Universal Robots PolyScope program: step5d_strict_rnn_autotune_v3_r022.urp

Program step5d_strict_rnn_autotune_v3_r022 (installation=default directory=/programs/andyl/kunwei/step5 createdIn=5.11.9.1010452 lastSavedIn=5.11.9.1010452 robotSerialNumber=20225200364)
Calibrated DH parameters: a=[0.00002, -0.569483, -0.54992, -0.00001, -0.000036, 0]; d=[0.180894, -146.691669, 192.918669, -46.053088, 0.119778, 0.115602]; alpha=[1.571425, -0.001534, 0.003359, 1.568739, -1.571477, 0]; deltaTheta=[0, 0.376258, -0.101074, -0.275185, -0.000002, 0]
Robot Program (runOnlyOnce=true)
  Script file /programs/andyl/kunwei/step5/step5d_strict_rnn_autotune_v3_r022.script
    | # VERSION: 2026-07-25T163424Z
    | # RELEASE_STAGE_ID: step5d_strict_rnn_autotune_v3_r022
    | # CONTROL_PROFILE_ID: step5d_strict_rnn_autotune_v1
    | # TP_PROGRAM_ID: step5d_strict_rnn_autotune_v3_r022
    | # PHYSICAL_PRIOR_SHA256: c8019aee2c293746e1edb23097aeab1d7dfb1b8dee09df10ce568fb634f47c9f
    | # PARENT_AUTOTUNE_V1_RENDERED_SHA256: eca2c7acaa878b1944c24b46c823ed64ffc0fb9e8658021dfd863a9f624f6676
    | # TP_RUNTIME_IDENTITY_INT: protocol_version=35 digest_hi=36 digest_lo=37
    | global codex_step5d_runtime_protocol_version = 1
    | global codex_step5d_runtime_digest_hi = 1956245643
    | global codex_step5d_runtime_digest_lo = 189200615
    | 
    | def codex_step5d_publish_runtime_identity():
    |   write_output_integer_register(35, codex_step5d_runtime_protocol_version)
    |   write_output_integer_register(36, codex_step5d_runtime_digest_hi)
    |   write_output_integer_register(37, codex_step5d_runtime_digest_lo)
    | end
    | 
    | # Step5d strict RNN ablation v35.
    | # VERSION: 2026-07-15T0204HKT_STEP5D_STRICT_RNN_ABLATION_V35_QUOTA_SAFE_SCHED_OTHER_ACCEL_0P1
    | # GENERATED_AT_LOCAL: 2026-07-15T02:04:25+08:00
    | # ENTRY_XY_M: [0.487795411, 0.129326793]
    | # SAFE_FRAME_SOURCE: config/step5_safe_frame.json from confirmed drag-teach start/mid/end.
    | # NO_SCALE_POLICY: Step5 table frame uses rotation+translation only.
    | # X_GUARD: guard_line=0.488878434 m, path_max_x=0.487795411 m.
    | # TARGET_ROTVEC_RAD: [-3.044172198, -0.130573165, -0.202188631]
    | # PURPOSE: v35 contact search with Stage22/24 gravity-down pre-contact posture, first-contact normal latch, no lift/25.2 attitude cycle and no second contact search, 25.3 bridge deadband acquire into the 5.0-22.0N filtered preload window with 3.0-25.0N raw sanity and bridge-time preload parameter channel, 25.95 register clear barrier, then v35 Step5d ablation Stage25.0 layout-524-only speedj strict RNN live candidate for 60 s.
    | # FLOW_TABLE: STEP5_FLOW.md
    | # STEP5_STAGE_ID: step5d_strict_rnn_autotune_v3
    | # PARENT_V35_SHA256: 50894de5cdf74dd17309c829b904251a3da26613a4d73e93653f7c165f5fbbd0
    | # STEP5_TABLE_SOURCE: config/step5_stage_table.json
    | # TP_ROLE: layout524_speedj_executor_and_structural_guard_only; Step5d v35 accepts only bridge-computed strict RNN qdot; marker 524 is internal to the Stage25 joint packet.
    | # REGISTER_CONTRACT: Stage 25.3 is a no-motion structural handoff. Stage 25.95 requires bridge-cleared registers 37..47 before Stage 25.0. Stage 25.0 accepts only register 47=524.0; registers 37..42 are strict RNN qd0..qd5, 43 cmd_valid, 44 path_time_s. Layout 523.0 and Cartesian/DLS runtime commands are forbidden.
    | # PRECONTACT_POSE_CONTRACT: config/step_pose_contract_table.json pre_contact_search_gravity_down_v1; Stage22/24 TCP +Z targets base -Z using [pi,0,0].
    | # STAGE25_CONTACT_SAFETY: v35 bridge keeps 60N normal/100N force guards and 3.0Nm torque guard; speedj_rnn_live is the only future live command source; speedl_cartesian_oracle and speedj_dls_oracle are offline shadow/diagnostic only and must never be sent as runtime fallback.
    | # FORCE_FRAME_CONTRACT: UR_FORCE_FRAME_CONTRACT.md; reaction normal for load, approach normal for posture.
    | # STAGE25_V35_SCAFFOLD: v31_permissive_contact_frame_contract_layout524_60s
    | # STEP5_PATH_FORMULA: Step5 table stage step5_contact_cycloid_baseline_v1: local-basis x=0.015 * (0.1t - sin(0.1t)), y=0.015 * (1 - cos(0.1t)), duration=60s
    | # FIRST_CONTACT_Z_EVIDENCE: bridge_step4e_line_outerloop_v13_autowatch_20260609_141027 force jump at z=0.008044839 m; v16 cross-check z=0.007996174 m.
    | # AUTOTUNE_CONTROL: fixed tau=.35s, fixed dt=.002s, profile rate .010/.015/.020; normal_filter_alpha is not an active candidate dimension.
    | # SAFETY: raw normal guard 60 N, force norm guard 100 N, torque guard 3.0 Nm.
    | 
    | def codex_abs(x):
    |   if x < 0.0:
    |     return -x
    |   end
    |   return x
    | end
    | 
    | def codex_clamp(x, lo, hi):
    |   if x < lo:
    |     return lo
    |   elif x > hi:
    |     return hi
    |   end
    |   return x
    | end
    | 
    | def codex_wait_for_fresh_heartbeat(timeout_s):
    |   local t = 0.0
    |   local initial_heartbeat = read_input_float_register(26)
    |   local current_heartbeat = initial_heartbeat
    |   while t < timeout_s:
    |     current_heartbeat = read_input_float_register(26)
    |     write_output_float_register(26, current_heartbeat)
    |     if read_input_float_register(27) > 0.5 and current_heartbeat != initial_heartbeat:
    |       return True
    |     end
    |     sync()
    |     t = t + get_steptime()
    |   end
    |   return False
    | end
    | 
    | def codex_wait_for_rezero_complete(timeout_s):
    |   local t = 0.0
    |   local initial_heartbeat = read_input_float_register(26)
    |   local current_heartbeat = initial_heartbeat
    |   local saw_sensor_not_ready = False
    |   while t < timeout_s:
    |     current_heartbeat = read_input_float_register(26)
    |     write_output_float_register(26, current_heartbeat)
    |     if read_input_float_register(27) < 0.5:
    |       saw_sensor_not_ready = True
    |     elif saw_sensor_not_ready and read_input_float_register(27) > 0.5 and current_heartbeat != initial_heartbeat:
    |       return True
    |     end
    |     sync()
    |     t = t + get_steptime()
    |   end
    |   return False
    | end
    | 
    | def codex_step4e_guard_stop_reason():
    |   local normal_force = read_input_float_register(24)
    |   local force_norm = read_input_float_register(25)
    |   local sensor_ok = read_input_float_register(27)
    |   local stop_request = read_input_float_register(28)
    |   local torque_norm = read_input_float_register(30)
    |   if sensor_ok < 0.5:
    |     return 3.0
    |   elif stop_request > 0.5:
    |     return 4.0
    |   elif codex_abs(normal_force) > 60.0:
    |     return 5.0
    |   elif force_norm > 100.0:
    |     return 6.0
    |   elif torque_norm > 3.0:
    |     return 7.0
    |   end
    |   return 0.0
    | end
    | 
    | def codex_should_auto_home(stop_reason):
    |   if stop_reason == 1.0:
    |     return True
    |   elif stop_reason == 2.0:
    |     # Transport/heartbeat loss may follow a protective stop; never auto-home.
    |     return False
    |   elif stop_reason == 4.0:
    |     return True
    |   elif stop_reason == 5.0:
    |     return True
    |   elif stop_reason == 6.0:
    |     return True
    |   elif stop_reason == 7.0:
    |     return True
    |   elif stop_reason == 8.0:
    |     return True
    |   elif stop_reason == 9.0:
    |     return True
    |   elif stop_reason == 10.0:
    |     return True
    |   elif stop_reason == 12.0:
    |     return True
    |   elif stop_reason == 13.0:
    |     return True
    |   elif stop_reason == 14.0:
    |     return True
    |   elif stop_reason == 17.0:
    |     # Reserved unsafe-entry/safety interruption reason; never auto-home.
    |     return False
    |   end
    |   return False
    | end
    | 
    | def codex_echo_basic(stop_reason):
    |   write_output_float_register(24, read_input_float_register(24))
    |   write_output_float_register(25, read_input_float_register(25))
    |   write_output_float_register(26, read_input_float_register(26))
    |   write_output_float_register(27, read_input_float_register(27))
    |   write_output_float_register(28, read_input_float_register(28))
    |   write_output_float_register(29, read_input_float_register(29))
    |   write_output_float_register(30, stop_reason)
    | end
    | 
    | def codex_echo_step4e(stop_reason):
    |   codex_echo_basic(stop_reason)
    |   write_output_float_register(31, read_input_float_register(44))
    |   write_output_float_register(32, read_input_float_register(45))
    |   write_output_float_register(33, read_input_float_register(39))
    |   write_output_float_register(36, read_input_float_register(37))
    |   write_output_float_register(37, read_input_float_register(38))
    |   write_output_float_register(38, read_input_float_register(39))
    |   write_output_float_register(39, read_input_float_register(40))
    |   write_output_float_register(40, read_input_float_register(41))
    |   write_output_float_register(41, read_input_float_register(42))
    |   write_output_float_register(42, read_input_float_register(43))
    |   write_output_float_register(43, read_input_float_register(44))
    |   write_output_float_register(44, read_input_float_register(45))
    |   write_output_float_register(45, read_input_float_register(46))
    |   write_output_float_register(46, read_input_float_register(47))
    | end
    | 
    | 
    | def codex_wait_for_cmd_valid(stage_code, timeout_s):
    |   local t = 0.0
    |   local last_heartbeat = read_input_float_register(26)
    |   local stale_s = 0.0
    |   while t < timeout_s:
    |     write_output_float_register(35, stage_code)
    |     local heartbeat = read_input_float_register(26)
    |     if heartbeat == last_heartbeat:
    |       stale_s = stale_s + get_steptime()
    |     else:
    |       stale_s = 0.0
    |       last_heartbeat = heartbeat
    |     end
    |     codex_echo_step4e(0.0)
    |     if stale_s > 0.100:
    |       return 2.0
    |     end
    |     local guard_reason = codex_step4e_guard_stop_reason()
    |     if guard_reason != 0.0:
    |       return guard_reason
    |     end
    |     if read_input_float_register(43) >= 0.5:
    |       return 0.0
    |     end
    |     sync()
    |     t = t + get_steptime()
    |   end
    |   return 12.0
    | end
    | 
    | 
    | def codex_wait_for_stage_linear_zero(stage_code, timeout_s):
    |   local t = 0.0
    |   local last_heartbeat = read_input_float_register(26)
    |   local stale_s = 0.0
    |   while t < timeout_s:
    |     write_output_float_register(35, stage_code)
    |     local heartbeat = read_input_float_register(26)
    |     if heartbeat == last_heartbeat:
    |       stale_s = stale_s + get_steptime()
    |     else:
    |       stale_s = 0.0
    |       last_heartbeat = heartbeat
    |     end
    |     codex_echo_step4e(0.0)
    |     if stale_s > 0.100:
    |       return 2.0
    |     end
    |     local guard_reason = codex_step4e_guard_stop_reason()
    |     if guard_reason != 0.0:
    |       return guard_reason
    |     end
    |     if read_input_float_register(43) >= 0.5 and codex_abs(read_input_float_register(37)) <= 0.000001 and codex_abs(read_input_float_register(38)) <= 0.000001 and codex_abs(read_input_float_register(39)) <= 0.000001:
    |       return 0.0
    |     end
    |     sync()
    |     t = t + get_steptime()
    |   end
    |   return 12.0
    | end
    | 
    | def codex_step5d_down_search(search_stage, near_stage, max_search_down_m, search_near_start_depth_m, search_runtime_limit_s, search_far_speed_m_s, search_near_speed_m_s):
    |   local stop_reason = 0.0
    |   local search_accel_m_s2 = 0.300
    |   local search_hold_s = 0.002
    |   local stale_limit_s = 0.100
    |   local search_start = get_actual_tcp_pose()
    |   local last_heartbeat = read_input_float_register(26)
    |   local stale_s = 0.0
    |   local t = 0.0
    |   while stop_reason == 0.0:
    |     local heartbeat = read_input_float_register(26)
    |     local normal_force = read_input_float_register(24)
    |     local force_norm = read_input_float_register(25)
    |     local pose_now = get_actual_tcp_pose()
    |     local search_depth_m = search_start[2] - pose_now[2]
    |     if heartbeat == last_heartbeat:
    |       stale_s = stale_s + get_steptime()
    |     else:
    |       stale_s = 0.0
    |       last_heartbeat = heartbeat
    |     end
    |     if normal_force <= -1.0 or force_norm > 1.5:
    |       stop_reason = 11.0
    |       if search_depth_m < search_near_start_depth_m:
    |         write_output_float_register(35, search_stage)
    |       else:
    |         write_output_float_register(35, near_stage)
    |       end
    |       codex_echo_step4e(stop_reason)
    |     elif stale_s > stale_limit_s:
    |       stop_reason = 2.0
    |     else:
    |       stop_reason = codex_step4e_guard_stop_reason()
    |     end
    |     if stop_reason == 0.0:
    |       if search_depth_m >= max_search_down_m:
    |         stop_reason = 8.0
    |       elif t >= search_runtime_limit_s:
    |         stop_reason = 10.0
    |       else:
    |         if search_depth_m < search_near_start_depth_m:
    |           write_output_float_register(35, search_stage)
    |           codex_echo_step4e(stop_reason)
    |           speedl([0.0, 0.0, search_far_speed_m_s, 0.0, 0.0, 0.0], search_accel_m_s2, search_hold_s)
    |         else:
    |           write_output_float_register(35, near_stage)
    |           codex_echo_step4e(stop_reason)
    |           speedl([0.0, 0.0, search_near_speed_m_s, 0.0, 0.0, 0.0], search_accel_m_s2, search_hold_s)
    |         end
    |         t = t + get_steptime()
    |       end
    |     end
    |   end
    |   stopl(0.1)
    |   return stop_reason
    | end
    | 
    | def codex_step5d_autotune_trial_v1(campaign_home_pose, tp_speedj_accel_rad_s2, batch_row_index):
    |   local stop_reason = 0.0
    |   local home_pose = campaign_home_pose
    |   local entry_x = 0.487834547
    |   local entry_y = 0.129337053
    |   local precontact_z = 0.022863519
    |   local minimum_start_above_entry_m = 0.010000000
    |   # PRECONTACT_POSE_PRIOR_ID: step5d_v3_physical_prior_contact_0p1_20260719; completed contact-plus-0.1s robust pose plus clearance before guarded search.
    |   local target_rx = 3.120752062
    |   local target_ry = 0.000000000
    |   local target_rz = 0.068626833
    |   local line_accel_m_s2 = 0.300
    |   local line_hold_s = 0.002
    |   local line_runtime_limit_s = 75.000
    |   local line_success_progress_m = 60.000000000
    |   local end_hold_required_s = 0.100
    |   local end_hold_s = 0.0
    |   local max_cmd_angular_xy_rad_s = 0.120
    |   local cmd_valid_grace_s = 0.250
    |   local cmd_valid_loss_limit_s = 0.100
    |   local cmd_invalid_s = 0.0
    |   local saw_cmd_valid = 0
    |   local short_retract_z_m = 0.010
    |   local short_retract_speed_m_s = 0.040
    |   local home_return_speed_m_s = 0.050
    |   local final_progress_m = 0.0
    | 
    |   textmsg("codex step4e version 2026-07-15T0204HKT_STEP5D_STRICT_RNN_ABLATION_V35_QUOTA_SAFE_SCHED_OTHER_ACCEL_0P1 start step5d_strict_rnn_ablation_v35")
    |   write_output_float_register(34, 0.0)
    |   write_output_float_register(35, 20.0)
    |   codex_echo_step4e(0.0)
    |   if not codex_wait_for_fresh_heartbeat(60.0):
    |     stop_reason = 3.0
    |   end
    | 
    |   if stop_reason == 0.0:
    |     local p_current = get_actual_tcp_pose()
    |     local expected_home_orientation = p[p_current[0], p_current[1], p_current[2], target_rx, target_ry, target_rz]
    |     local home_orientation_delta = pose_trans(pose_inv(expected_home_orientation), p_current)
    |     local home_orientation_error_rad = sqrt(home_orientation_delta[3] * home_orientation_delta[3] + home_orientation_delta[4] * home_orientation_delta[4] + home_orientation_delta[5] * home_orientation_delta[5])
    |     if p_current[2] < precontact_z + minimum_start_above_entry_m or home_orientation_error_rad > 0.035:
    |       return 17.0
    |     else:
    |       write_output_float_register(35, 22.0)
    |       local entry_xy_pose = p[entry_x, entry_y, p_current[2], target_rx, target_ry, target_rz]
    |       local entry_precontact_pose = p[entry_x, entry_y, precontact_z, target_rx, target_ry, target_rz]
    |       codex_echo_step4e(stop_reason)
    |       movel(entry_xy_pose, a=0.135, v=0.090, r=0.0)
    |       stopl(0.1)
    |       movel(entry_precontact_pose, a=0.060, v=0.040, r=0.0)
    |       stopl(0.1)
    |       sleep(0.20)
    |     end
    |     write_output_float_register(35, 23.0)
    |     codex_echo_step4e(stop_reason)
    |     write_output_float_register(34, 1.0)
    |     if not codex_wait_for_rezero_complete(5.0):
    |       stop_reason = 14.0
    |     end
    |     if stop_reason == 0.0:
    |       sleep(0.20)
    |       stop_reason = codex_step4e_guard_stop_reason()
    |     end
    |   end
    | 
    |   if stop_reason == 0.0:
    |     local first_contact_z_m = 0.008044839
    |     local first_near_start_z_m = first_contact_z_m + 0.020
    |     local first_max_end_z_m = first_contact_z_m - 0.004
    |     local first_search_start_pose = get_actual_tcp_pose()
    |     local first_search_near_start_depth_m = first_search_start_pose[2] - first_near_start_z_m
    |     local first_search_max_down_m = first_search_start_pose[2] - first_max_end_z_m
    |     if first_search_near_start_depth_m < 0.0:
    |       first_search_near_start_depth_m = 0.0
    |     end
    |     if first_search_max_down_m < 0.020:
    |       first_search_max_down_m = 0.020
    |     end
    |     if first_search_max_down_m < first_search_near_start_depth_m + 0.010:
    |       first_search_max_down_m = first_search_near_start_depth_m + 0.010
    |     end
    |     stop_reason = codex_step5d_down_search(24.0, 24.2, first_search_max_down_m, first_search_near_start_depth_m, 40.000, -0.03375, -0.0025)
    |     if stop_reason == 11.0:
    |       stop_reason = 0.0
    |     end
    |   end
    | 
    |   if stop_reason == 0.0:
    |     write_output_float_register(35, 25.05)
    |     stop_reason = codex_wait_for_cmd_valid(25.05, 1.000)
    |   end
    | 
    |   if stop_reason == 0.0:
    |     write_output_float_register(35, 25.15)
    |     codex_echo_step4e(stop_reason)
    |     sync()
    |   end
    | 
    |   if stop_reason == 0.0:
    |     write_output_float_register(35, 25.3)
    |     local last_heartbeat_entry = read_input_float_register(26)
    |     local stale_s_entry = 0.0
    |     local t_entry = 0.0
    |     local line_entry_s = 0.0
    |     local line_entry_default_required_s = 0.000
    |     local line_entry_default_timeout_s = 60.000
    |     local line_entry_default_normal_load_min_n = 5.000
    |     local line_entry_default_normal_load_max_n = 22.000
    |     local line_entry_default_force_norm_max_n = 100.000
    |     local line_entry_recovery_normal_load_min_n = 0.000
    |     local line_entry_recovery_normal_load_max_n = 100.000
    |     local line_entry_force_norm_stop_n = 100.000
    |     local line_entry_cmd_limit_m_s = 0.003
    |     local line_entry_param_valid_code = 521.000
    |     saw_cmd_valid = 0
    |     cmd_invalid_s = 0.0
    |     while stop_reason == 0.0:
    |       local heartbeat_entry = read_input_float_register(26)
    |       local cmd_valid = read_input_float_register(43)
    |       local cmd_vx = read_input_float_register(37)
    |       local cmd_vy = read_input_float_register(38)
    |       local cmd_vz = read_input_float_register(39)
    |       local target_force = read_input_float_register(29)
    |       local force_error = read_input_float_register(45)
    |       local normal_load = target_force - force_error
    |       local force_norm = read_input_float_register(25)
    |       local loop_dt = get_steptime()
    |       local line_entry_required_s = line_entry_default_required_s
    |       local line_entry_timeout_s = line_entry_default_timeout_s
    |       local line_entry_normal_load_min_n = line_entry_default_normal_load_min_n
    |       local line_entry_normal_load_max_n = line_entry_default_normal_load_max_n
    |       local line_entry_force_norm_max_n = line_entry_default_force_norm_max_n
    |       local line_entry_param_valid = read_input_float_register(47)
    |       if codex_abs(line_entry_param_valid - line_entry_param_valid_code) < 0.001:
    |         local candidate_min_n = read_input_float_register(40)
    |         local candidate_max_n = read_input_float_register(41)
    |         local candidate_force_norm_max_n = read_input_float_register(42)
    |         local candidate_required_s = read_input_float_register(44)
    |         local candidate_timeout_s = read_input_float_register(46)
    |         if candidate_min_n >= 0.0 and candidate_max_n >= candidate_min_n and candidate_force_norm_max_n > 0.0 and candidate_force_norm_max_n <= line_entry_force_norm_stop_n and candidate_required_s >= 0.0 and candidate_timeout_s > candidate_required_s:
    |           line_entry_normal_load_min_n = candidate_min_n
    |           line_entry_normal_load_max_n = candidate_max_n
    |           line_entry_force_norm_max_n = candidate_force_norm_max_n
    |           line_entry_required_s = candidate_required_s
    |           line_entry_timeout_s = candidate_timeout_s
    |         end
    |       end
    |       if cmd_valid >= 0.5:
    |         saw_cmd_valid = 1
    |         cmd_invalid_s = 0.0
    |       else:
    |         cmd_invalid_s = cmd_invalid_s + loop_dt
    |       end
    |       if heartbeat_entry == last_heartbeat_entry:
    |         stale_s_entry = stale_s_entry + loop_dt
    |       else:
    |         stale_s_entry = 0.0
    |         last_heartbeat_entry = heartbeat_entry
    |       end
    |       t_entry = t_entry + loop_dt
    |       if cmd_valid >= 0.5:
    |         line_entry_s = line_entry_s + loop_dt
    |       else:
    |         line_entry_s = 0.0
    |       end
    |       codex_echo_step4e(stop_reason)
    |       if stale_s_entry > 1.000:
    |         stop_reason = 2.0
    |       else:
    |         stop_reason = codex_step4e_guard_stop_reason()
    |       end
    |       if stop_reason == 0.0:
    |         if line_entry_s >= line_entry_required_s:
    |           stop_reason = 16.0
    |         elif cmd_valid < 0.5:
    |           if saw_cmd_valid == 0 and t_entry < cmd_valid_grace_s:
    |             sync()
    |           elif saw_cmd_valid == 1 and cmd_invalid_s <= cmd_valid_loss_limit_s:
    |             sync()
    |           else:
    |             stop_reason = 12.0
    |           end
    |         elif t_entry >= line_entry_timeout_s:
    |           stop_reason = 12.0
    |         else:
    |           sync()
    |         end
    |       end
    |     end
    |     stopl(0.1)
    |     if stop_reason == 16.0:
    |       stop_reason = 0.0
    |       saw_cmd_valid = 0
    |       cmd_invalid_s = 0.0
    |       end_hold_s = 0.0
    |       write_output_float_register(35, 25.95)
    |       local register_clear_required_s = 0.006
    |       local register_clear_timeout_s = 1.000
    |       local register_clear_s = 0.0
    |       local register_clear_t = 0.0
    |       local register_clear_zero_tol = 0.000500
    |       local last_heartbeat_clear = read_input_float_register(26)
    |       local stale_s_clear = 0.0
    |       while stop_reason == 0.0 and register_clear_s < register_clear_required_s and register_clear_t < register_clear_timeout_s:
    |         local heartbeat_clear = read_input_float_register(26)
    |         local clear_cmd_valid = read_input_float_register(43)
    |         local clear_reg0 = read_input_float_register(37)
    |         local clear_reg1 = read_input_float_register(38)
    |         local clear_reg2 = read_input_float_register(39)
    |         local clear_reg3 = read_input_float_register(40)
    |         local clear_reg4 = read_input_float_register(41)
    |         local clear_reg5 = read_input_float_register(42)
    |         local clear_layout_tag = read_input_float_register(47)
    |         local loop_dt = get_steptime()
    |         if heartbeat_clear == last_heartbeat_clear:
    |           stale_s_clear = stale_s_clear + loop_dt
    |         else:
    |           stale_s_clear = 0.0
    |           last_heartbeat_clear = heartbeat_clear
    |         end
    |         register_clear_t = register_clear_t + loop_dt
    |         codex_echo_step4e(stop_reason)
    |         if stale_s_clear > 1.000:
    |           stop_reason = 2.0
    |         else:
    |           stop_reason = codex_step4e_guard_stop_reason()
    |         end
    |         if stop_reason == 0.0:
    |           if clear_cmd_valid < 0.5 and codex_abs(clear_layout_tag - line_entry_param_valid_code) >= 0.001 and codex_abs(clear_layout_tag - 523.000) >= 0.001 and codex_abs(clear_layout_tag - 524.000) >= 0.001 and codex_abs(clear_reg0) <= register_clear_zero_tol and codex_abs(clear_reg1) <= register_clear_zero_tol and codex_abs(clear_reg2) <= register_clear_zero_tol and codex_abs(clear_reg3) <= register_clear_zero_tol and codex_abs(clear_reg4) <= register_clear_zero_tol and codex_abs(clear_reg5) <= register_clear_zero_tol:
    |             register_clear_s = register_clear_s + loop_dt
    |           else:
    |             register_clear_s = 0.0
    |           end
    |           sync()
    |         end
    |       end
    |       if stop_reason == 0.0 and register_clear_s < register_clear_required_s:
    |         stop_reason = 12.0
    |       end
    |     end
    |   end
    | 
    |   if stop_reason == 0.0:
    |     write_output_float_register(35, 25.0)
    |     local last_heartbeat2 = read_input_float_register(26)
    |     local stale_s2 = 0.0
    |     local t2 = 0.0
    |     local qdot_cap_rad_s = 0.500
    |     local cartesian_linear_cap_m_s = 1.000
    |     local cartesian_angular_cap_rad_s = 1.000
    |     local cartesian_accel_m_s2 = 0.050
    |     local joint_accel_rad_s2 = tp_speedj_accel_rad_s2
    |     local cartesian_layout_code = 523.000
    |     local joint_layout_code = 524.000
    |     local stage25_have_accepted_command = False
    |     # STAGE25_CADENCE_CONSUMPTION: output register 47 is 1 only when this
    |     # TP loop accepts a current Stage25 command packet and reaches speedl/speedj.
    |     while stop_reason == 0.0:
    |       local heartbeat2 = read_input_float_register(26)
    |       local cmd_valid = read_input_float_register(43)
    |       local progress_s = read_input_float_register(44)
    |       local stage25_layout_tag = read_input_float_register(47)
    |       local stage25_command_consumed = 0
    |       local cartesian_layout_ok = codex_abs(stage25_layout_tag - cartesian_layout_code) < 0.001
    |       local joint_layout_ok = codex_abs(stage25_layout_tag - joint_layout_code) < 0.001
    |       local cmd_qd0 = read_input_float_register(37)
    |       local cmd_qd1 = read_input_float_register(38)
    |       local cmd_qd2 = read_input_float_register(39)
    |       local cmd_qd3 = read_input_float_register(40)
    |       local cmd_qd4 = read_input_float_register(41)
    |       local cmd_qd5 = read_input_float_register(42)
    |       local cmd_vx = cmd_qd0
    |       local cmd_vy = cmd_qd1
    |       local cmd_vz = cmd_qd2
    |       local cmd_wx = cmd_qd3
    |       local cmd_wy = cmd_qd4
    |       local cmd_wz = cmd_qd5
    |       local loop_dt = get_steptime()
    |       local heartbeat_fresh = False
    |       final_progress_m = progress_s
    |       if cmd_valid >= 0.5 and joint_layout_ok:
    |         saw_cmd_valid = 1
    |         cmd_invalid_s = 0.0
    |       else:
    |         cmd_invalid_s = cmd_invalid_s + loop_dt
    |       end
    |       if heartbeat2 == last_heartbeat2:
    |         stale_s2 = stale_s2 + loop_dt
    |       else:
    |         stale_s2 = 0.0
    |         last_heartbeat2 = heartbeat2
    |         heartbeat_fresh = True
    |       end
    |       t2 = t2 + loop_dt
    |       if progress_s >= line_success_progress_m:
    |         end_hold_s = end_hold_s + loop_dt
    |       else:
    |         end_hold_s = 0.0
    |       end
    |       codex_echo_step4e(stop_reason)
    |       if stale_s2 > 1.000:
    |         stop_reason = 2.0
    |       else:
    |         stop_reason = codex_step4e_guard_stop_reason()
    |       end
    |       if stop_reason == 0.0:
    |         # DEADLINE_OVERRUN_LAST_COMMAND_HOLD: bounded zero-order hold.
    |         if not heartbeat_fresh:
    |           if stage25_have_accepted_command and cmd_valid >= 0.5 and joint_layout_ok and codex_abs(cmd_qd0) <= qdot_cap_rad_s and codex_abs(cmd_qd1) <= qdot_cap_rad_s and codex_abs(cmd_qd2) <= qdot_cap_rad_s and codex_abs(cmd_qd3) <= qdot_cap_rad_s and codex_abs(cmd_qd4) <= qdot_cap_rad_s and codex_abs(cmd_qd5) <= qdot_cap_rad_s:
    |             stage25_command_consumed = 1
    |             write_output_float_register(47, stage25_command_consumed)
    |             speedj([cmd_qd0, cmd_qd1, cmd_qd2, cmd_qd3, cmd_qd4, cmd_qd5], joint_accel_rad_s2, line_hold_s)
    |           else:
    |             write_output_float_register(47, stage25_command_consumed)
    |             sync()
    |           end
    |         elif cmd_valid < 0.5 or not joint_layout_ok:
    |           write_output_float_register(47, stage25_command_consumed)
    |           if saw_cmd_valid == 0 and t2 < cmd_valid_grace_s:
    |             sync()
    |           elif saw_cmd_valid == 1 and cmd_invalid_s <= cmd_valid_loss_limit_s:
    |             sync()
    |           else:
    |             stop_reason = 12.0
    |           end
    |         elif joint_layout_ok and (codex_abs(cmd_qd0) > qdot_cap_rad_s or codex_abs(cmd_qd1) > qdot_cap_rad_s or codex_abs(cmd_qd2) > qdot_cap_rad_s or codex_abs(cmd_qd3) > qdot_cap_rad_s or codex_abs(cmd_qd4) > qdot_cap_rad_s or codex_abs(cmd_qd5) > qdot_cap_rad_s):
    |           write_output_float_register(47, stage25_command_consumed)
    |           stop_reason = 13.0
    |         elif end_hold_s >= end_hold_required_s:
    |           write_output_float_register(47, stage25_command_consumed)
    |           stop_reason = 1.0
    |         elif t2 >= line_runtime_limit_s:
    |           write_output_float_register(47, stage25_command_consumed)
    |           stop_reason = 10.0
    |         else:
    |           stage25_have_accepted_command = True
    |           stage25_command_consumed = 1
    |           write_output_float_register(47, stage25_command_consumed)
    |           speedj([cmd_qd0, cmd_qd1, cmd_qd2, cmd_qd3, cmd_qd4, cmd_qd5], joint_accel_rad_s2, line_hold_s)
    |         end
    |       end
    |     end
    |     stopj(0.3)
    |     stopl(0.1)
    |   end
    | 
    |   write_output_float_register(30, stop_reason)
    |   write_output_float_register(31, final_progress_m)
    |   write_output_float_register(35, 29.0)
    |   textmsg("codex step4e version 2026-07-15T0204HKT_STEP5D_STRICT_RNN_ABLATION_V35_QUOTA_SAFE_SCHED_OTHER_ACCEL_0P1 stop reason:", stop_reason)
    |   return stop_reason
    | end
    | 
    | # STEP5D_AUTOTUNE_CONTINUOUS_TP: every trial returns to the captured campaign home.
    | # Immutable bundle cold-read precedes each rolling next ARM; no ACK command is active.
    | # HOST_TO_TP_INT: epoch=24 trial=25 command=26 token=27 profile=28 sequence=29 batch_row=30 logical_batch=31
    | # TP_TO_HOST_INT: epoch=24 trial=25 state=26 token=27 reason=28 profile=29 consumed_sequence=30 batch_row=31 return_kind=32 guard_mask=33 logical_batch=34
    | # PROFILE_ID: hundreds=normal-rate level; tens=host-slew level; ones=TP accel level
    | # NETWORK_PROFILE_LEVELS: normal=1..3 (.010/.015/.020); host/TP=1..3 (.1/.2/.5)
    | # PROFILE_NORMAL_LEVELS: 1=.010, 2=.015, 3=.020, 5=.050, 6=.100 rad/s;
    | # level 4 (.030 rad/s) is offline_only and must never reach this TP
    | # TP_ACCEL_LEVEL: 1=.1 rad/s^2, 2=.2 rad/s^2, 3=.5 rad/s^2
    | # STOP_CONTRACT: integer STOP is polled only in stationary ready states; during RUN
    | # the frozen trial consumes the legacy float stop_request safety carrier.
    | 
    | global codex_autotune_batch_row_echo = 0
    | global codex_autotune_return_kind_echo = 0
    | global codex_autotune_return_guard_mask = 0
    | global codex_autotune_return_observer_active = False
    | global codex_autotune_return_segment_id = 0
    | global codex_autotune_return_current_angular_speed_rad_s = 0.0
    | global codex_autotune_return_current_angular_accel_rad_s2 = 0.0
    | global codex_autotune_return_max_angular_speed_rad_s = 0.0
    | global codex_autotune_return_max_angular_accel_rad_s2 = 0.0
    | global codex_autotune_return_max_sample_gap_s = 0.0
    | global codex_autotune_logical_batch_sequence_echo = 0
    | 
    | def codex_autotune_norm3(x, y, z):
    |   return sqrt(x * x + y * y + z * z)
    | end
    | 
    | thread codex_autotune_return_telemetry_observer():
    |   local have_controller_time_sample = False
    |   local have_angular_sample = False
    |   local last_wx = 0.0
    |   local last_wy = 0.0
    |   local last_wz = 0.0
    |   local controller_clock = time()
    |   local last_controller_time_s = controller_clock.sec + controller_clock.nanosec / 1000000000.0
    |   while codex_autotune_return_observer_active:
    |     controller_clock = time()
    |     local controller_time_s = controller_clock.sec + controller_clock.nanosec / 1000000000.0
    |     local loop_dt = controller_time_s - last_controller_time_s
    |     last_controller_time_s = controller_time_s
    |     local tcp_speed = get_actual_tcp_speed()
    |     local angular_speed_rad_s = codex_autotune_norm3(tcp_speed[3], tcp_speed[4], tcp_speed[5])
    |     local angular_accel_rad_s2 = 0.0
    |     if have_controller_time_sample and have_angular_sample and loop_dt > 0.0:
    |       local angular_filter_alpha = loop_dt / (0.020 + loop_dt)
    |       local filtered_wx = last_wx + angular_filter_alpha * (tcp_speed[3] - last_wx)
    |       local filtered_wy = last_wy + angular_filter_alpha * (tcp_speed[4] - last_wy)
    |       local filtered_wz = last_wz + angular_filter_alpha * (tcp_speed[5] - last_wz)
    |       angular_accel_rad_s2 = codex_autotune_norm3(filtered_wx - last_wx, filtered_wy - last_wy, filtered_wz - last_wz) / loop_dt
    |       last_wx = filtered_wx
    |       last_wy = filtered_wy
    |       last_wz = filtered_wz
    |     else:
    |       last_wx = tcp_speed[3]
    |       last_wy = tcp_speed[4]
    |       last_wz = tcp_speed[5]
    |     end
    |     have_angular_sample = True
    |     codex_autotune_return_current_angular_speed_rad_s = angular_speed_rad_s
    |     codex_autotune_return_current_angular_accel_rad_s2 = angular_accel_rad_s2
    |     if angular_speed_rad_s > codex_autotune_return_max_angular_speed_rad_s:
    |       codex_autotune_return_max_angular_speed_rad_s = angular_speed_rad_s
    |     end
    |     if angular_accel_rad_s2 > codex_autotune_return_max_angular_accel_rad_s2:
    |       codex_autotune_return_max_angular_accel_rad_s2 = angular_accel_rad_s2
    |     end
    |     if have_controller_time_sample and loop_dt > codex_autotune_return_max_sample_gap_s:
    |       codex_autotune_return_max_sample_gap_s = loop_dt
    |     end
    |     have_controller_time_sample = True
    |     sync()
    |   end
    | end
    | 
    | def codex_autotune_latch_return_telemetry():
    |   write_output_float_register(35, 40.3)
    |   write_output_float_register(39, 3.0)
    |   write_output_float_register(40, codex_autotune_return_current_angular_speed_rad_s)
    |   write_output_float_register(41, codex_autotune_return_current_angular_accel_rad_s2)
    |   write_output_float_register(42, codex_autotune_return_max_angular_speed_rad_s)
    |   write_output_float_register(43, codex_autotune_return_max_angular_accel_rad_s2)
    |   write_output_float_register(44, codex_autotune_return_max_sample_gap_s)
    | end
    | 
    | def codex_autotune_typed_target_verified(target_pose, campaign_home_q, require_home_q):
    |   local actual_pose = get_actual_tcp_pose()
    |   local delta_pose = pose_trans(pose_inv(target_pose), actual_pose)
    |   local position_error_m = sqrt(delta_pose[0] * delta_pose[0] + delta_pose[1] * delta_pose[1] + delta_pose[2] * delta_pose[2])
    |   local orientation_error_rad = sqrt(delta_pose[3] * delta_pose[3] + delta_pose[4] * delta_pose[4] + delta_pose[5] * delta_pose[5])
    |   local tcp_speed = get_actual_tcp_speed()
    |   local linear_speed_m_s = sqrt(tcp_speed[0] * tcp_speed[0] + tcp_speed[1] * tcp_speed[1] + tcp_speed[2] * tcp_speed[2])
    |   local angular_speed_rad_s = sqrt(tcp_speed[3] * tcp_speed[3] + tcp_speed[4] * tcp_speed[4] + tcp_speed[5] * tcp_speed[5])
    |   local actual_qd = get_actual_joint_speeds()
    |   local qd_max_rad_s = 0.0
    |   local qd_index = 0
    |   while qd_index < 6:
    |     if codex_abs(actual_qd[qd_index]) > qd_max_rad_s:
    |       qd_max_rad_s = codex_abs(actual_qd[qd_index])
    |     end
    |     qd_index = qd_index + 1
    |   end
    |   local home_q_ok = True
    |   if require_home_q:
    |     home_q_ok = codex_autotune_max_joint_error(campaign_home_q, get_actual_joint_positions()) <= 0.010
    |   end
    |   write_output_float_register(36, position_error_m)
    |   write_output_float_register(37, orientation_error_rad)
    |   write_output_float_register(38, qd_max_rad_s)
    |   return position_error_m <= 0.003 and orientation_error_rad <= 0.050 and linear_speed_m_s <= 0.001 and angular_speed_rad_s <= 0.010 and qd_max_rad_s <= 0.010 and home_q_ok
    | end
    | 
    | def codex_autotune_single_owner_return(batch_row_index, campaign_home_pose, campaign_home_q):
    |   local current_pose = get_actual_tcp_pose()
    |   local safe_z = 0.033
    |   local near_pose = p[0.487834547, 0.129337053, 0.022863519, 3.120752062, 0.000000000, 0.068626833]
    |   local target_pose = campaign_home_pose
    |   local require_home_q = True
    |   local rise_pose = p[current_pose[0], current_pose[1], safe_z, current_pose[3], current_pose[4], current_pose[5]]
    |   local transfer_pose = p[target_pose[0], target_pose[1], safe_z, target_pose[3], target_pose[4], target_pose[5]]
    |   codex_autotune_return_guard_mask = 0
    |   codex_autotune_return_segment_id = 0
    |   codex_autotune_return_current_angular_speed_rad_s = 0.0
    |   codex_autotune_return_current_angular_accel_rad_s2 = 0.0
    |   codex_autotune_return_max_angular_speed_rad_s = 0.0
    |   codex_autotune_return_max_angular_accel_rad_s2 = 0.0
    |   codex_autotune_return_max_sample_gap_s = 0.0
    |   codex_autotune_return_observer_active = True
    |   local return_observer_handle = run codex_autotune_return_telemetry_observer()
    |   codex_autotune_return_segment_id = 1
    |   movel(rise_pose, a=0.060, v=0.040, r=0.0)
    |   stopl(0.1)
    |   codex_autotune_return_segment_id = 2
    |   movel(transfer_pose, a=0.135, v=0.090, r=0.0)
    |   stopl(0.1)
    |   codex_autotune_return_segment_id = 3
    |   movel(target_pose, a=0.060, v=0.040, r=0.0)
    |   stopl(0.1)
    |   sleep(0.20)
    |   codex_autotune_return_observer_active = False
    |   sync()
    |   kill return_observer_handle
    |   if not codex_autotune_typed_target_verified(target_pose, campaign_home_q, require_home_q):
    |     return False
    |   end
    |   # The main TP thread is the only motion owner.  Host/controller closure
    |   # validates the seven typed safety signals after the sequential movel route.
    |   codex_autotune_return_guard_mask = 127
    |   codex_autotune_latch_return_telemetry()
    |   return True
    | end
    | 
    | def codex_autotune_write_state(campaign_epoch, trial_id, state, candidate_token, terminal_reason, execution_profile_id, consumed_command_seq):
    |   codex_step5d_publish_runtime_identity()
    |   write_output_integer_register(24, campaign_epoch)
    |   write_output_integer_register(25, trial_id)
    |   write_output_integer_register(27, candidate_token)
    |   write_output_integer_register(28, terminal_reason)
    |   write_output_integer_register(29, execution_profile_id)
    |   write_output_integer_register(31, codex_autotune_batch_row_echo)
    |   write_output_integer_register(32, codex_autotune_return_kind_echo)
    |   write_output_integer_register(33, codex_autotune_return_guard_mask)
    |   write_output_integer_register(34, codex_autotune_logical_batch_sequence_echo)
    |   write_output_integer_register(26, state)
    |   write_output_integer_register(30, consumed_command_seq)
    | end
    | 
    | def codex_autotune_speedj_accel(execution_profile_id):
    |   local accel_level = execution_profile_id - 10 * floor(execution_profile_id / 10.0)
    |   if accel_level == 1:
    |     return 0.100
    |   elif accel_level == 2:
    |     return 0.200
    |   elif accel_level == 3:
    |     return 0.500
    |   end
    |   return -1.000
    | end
    | 
    | def codex_autotune_network_profile_valid(execution_profile_id):
    |   local normal_level = floor(execution_profile_id / 100.0)
    |   local remainder = execution_profile_id - 100 * normal_level
    |   local host_slew_level = floor(remainder / 10.0)
    |   local tp_accel_level = remainder - 10 * host_slew_level
    |   return (normal_level >= 1 and normal_level <= 3 or normal_level == 5 or normal_level == 6) and host_slew_level >= 1 and host_slew_level <= 3 and tp_accel_level >= 1 and tp_accel_level <= 3
    | end
    | 
    | def codex_autotune_direct_terminal_state(stop_reason, batch_row_index):
    |   # Every local software guard is trial-local.  The controller owns hardware
    |   # safety stops; TP publishes READY_HOME_NEXT and waits for a fresh ARM.
    |   return 78
    | end
    | 
    | def codex_autotune_max_joint_error(home_q, actual_q):
    |   local maximum = 0.0
    |   local index = 0
    |   while index < 6:
    |     local error = codex_abs(home_q[index] - actual_q[index])
    |     if error > maximum:
    |       maximum = error
    |     end
    |     index = index + 1
    |   end
    |   return maximum
    | end
    | 
    | def codex_autotune_home_verified(campaign_home_pose, campaign_home_q):
    |   local actual_pose = get_actual_tcp_pose()
    |   local delta_pose = pose_trans(pose_inv(campaign_home_pose), actual_pose)
    |   local position_error_m = sqrt(delta_pose[0] * delta_pose[0] + delta_pose[1] * delta_pose[1] + delta_pose[2] * delta_pose[2])
    |   local orientation_error_rad = sqrt(delta_pose[3] * delta_pose[3] + delta_pose[4] * delta_pose[4] + delta_pose[5] * delta_pose[5])
    |   local joint_error_rad = codex_autotune_max_joint_error(campaign_home_q, get_actual_joint_positions())
    |   write_output_float_register(36, position_error_m)
    |   write_output_float_register(37, orientation_error_rad)
    |   write_output_float_register(38, joint_error_rad)
    |   return position_error_m <= 0.003 and orientation_error_rad <= 0.050 and joint_error_rad <= 0.010
    | end
    | 
    | def codex_autotune_publish_state_and_halt(campaign_epoch, trial_id, state, candidate_token, terminal_reason, execution_profile_id, consumed_command_seq):
    |   local publish_s = 0.0
    |   while publish_s < 0.100:
    |     codex_autotune_write_state(campaign_epoch, trial_id, state, candidate_token, terminal_reason, execution_profile_id, consumed_command_seq)
    |     sync()
    |     publish_s = publish_s + get_steptime()
    |   end
    |   halt
    | end
    | 
    | def codex_autotune_publish_fault_and_halt(campaign_epoch, trial_id, candidate_token, terminal_reason, execution_profile_id, consumed_command_seq):
    |   codex_autotune_publish_state_and_halt(campaign_epoch, trial_id, 90, candidate_token, terminal_reason, execution_profile_id, consumed_command_seq)
    | end
    | 
    | def codex_autotune_fault_forever(campaign_epoch, trial_id, candidate_token, terminal_reason, execution_profile_id, consumed_command_seq):
    |   while True:
    |     codex_autotune_write_state(campaign_epoch, trial_id, 75, candidate_token, terminal_reason, execution_profile_id, consumed_command_seq)
    |     sync()
    |   end
    | end
    | 
    | def codex_autotune_wait_for_external_home(campaign_epoch, trial_id, state, candidate_token, terminal_reason, execution_profile_id, consumed_command_seq, campaign_home_pose, campaign_home_q):
    |   # state 75 is WAITING_FOR_HARDWARE / WAIT_INFRA_READY.  This loop is
    |   # deliberately no-motion: only typed pose, Home-q, TCP-speed, and qdot
    |   # verification may release it to READY_HOME_NEXT.
    |   while True:
    |     codex_autotune_write_state(campaign_epoch, trial_id, 75, candidate_token, terminal_reason, execution_profile_id, consumed_command_seq)
    |     if codex_autotune_typed_target_verified(campaign_home_pose, campaign_home_q, True):
    |       return True
    |     end
    |     local next_command = read_input_integer_register(26)
    |     local next_sequence = read_input_integer_register(29)
    |     if next_command == 3 and next_sequence > consumed_command_seq:
    |       codex_autotune_publish_fault_and_halt(campaign_epoch, trial_id, candidate_token, 4, execution_profile_id, next_sequence)
    |     end
    |     sync()
    |   end
    | end
    | 
    | def codex_autotune_wait_for_arm(campaign_epoch, trial_id, state, candidate_token, terminal_reason, execution_profile_id, consumed_command_seq):
    |   while True:
    |     codex_autotune_write_state(campaign_epoch, trial_id, state, candidate_token, terminal_reason, execution_profile_id, consumed_command_seq)
    |     local next_command = read_input_integer_register(26)
    |     local next_sequence = read_input_integer_register(29)
    |     if next_command == 1 and next_sequence > consumed_command_seq:
    |       if state == 78 and (read_input_integer_register(24) <= 0 or read_input_integer_register(25) <= 0 or read_input_integer_register(27) <= 0 or read_input_integer_register(28) <= 0 or read_input_integer_register(30) < 1 or read_input_integer_register(30) > 5 or read_input_integer_register(31) <= 0 or not codex_autotune_network_profile_valid(read_input_integer_register(28))):
    |         codex_autotune_write_state(campaign_epoch, trial_id, 78, candidate_token, 13, execution_profile_id, consumed_command_seq)
    |       else:
    |         return True
    |       end
    |     elif state == 78 and next_command == 4 and next_sequence > consumed_command_seq and read_input_integer_register(24) == campaign_epoch and read_input_integer_register(25) == trial_id and read_input_integer_register(27) == candidate_token and read_input_integer_register(28) == execution_profile_id and read_input_integer_register(30) == codex_autotune_batch_row_echo and read_input_integer_register(31) == codex_autotune_logical_batch_sequence_echo:
    |       codex_autotune_publish_state_and_halt(campaign_epoch, trial_id, 77, candidate_token, terminal_reason, execution_profile_id, next_sequence)
    |     elif next_command == 3 and next_sequence > consumed_command_seq:
    |       codex_autotune_publish_fault_and_halt(campaign_epoch, trial_id, candidate_token, 4, execution_profile_id, next_sequence)
    |     elif trial_id > 0 and next_command == 2 and next_sequence > consumed_command_seq:
    |       # A stale/invalid local command is also trial-local; leave the TP
    |       # stationary in READY_HOME_NEXT until the next fresh ARM arrives.
    |       codex_autotune_write_state(campaign_epoch, trial_id, 78, candidate_token, 13, execution_profile_id, consumed_command_seq)
    |     end
    |     sync()
    |   end
    | end
    | 
    | def codex_step5d_strict_rnn_autotune_v3():
    |   # Campaign home is captured exactly once for the lifetime of this TP loop.
    |   local campaign_home_pose = get_actual_tcp_pose()
    |   local campaign_home_q = get_actual_joint_positions()
    |   local last_consumed_command_seq = 0
    |   codex_autotune_wait_for_arm(0, 0, 10, 0, 0, 0, 0)
    | 
    |   while True:
    |     local command = read_input_integer_register(26)
    |     local command_seq = read_input_integer_register(29)
    |     if command == 3 and command_seq > last_consumed_command_seq:
    |       last_consumed_command_seq = command_seq
    |       codex_autotune_publish_fault_and_halt(0, 0, 0, 4, 0, last_consumed_command_seq)
    |     elif command == 1 and command_seq > last_consumed_command_seq:
    |       local campaign_epoch = read_input_integer_register(24)
    |       local trial_id = read_input_integer_register(25)
    |       local candidate_token = read_input_integer_register(27)
    |       local execution_profile_id = read_input_integer_register(28)
    |       local batch_row_index = read_input_integer_register(30)
    |       local logical_batch_sequence = read_input_integer_register(31)
    |       local tp_speedj_accel_rad_s2 = codex_autotune_speedj_accel(execution_profile_id)
    |       last_consumed_command_seq = command_seq
    | 
    |       if campaign_epoch <= 0 or trial_id <= 0 or candidate_token <= 0 or execution_profile_id <= 0 or batch_row_index < 1 or batch_row_index > 5 or logical_batch_sequence <= 0 or not codex_autotune_network_profile_valid(execution_profile_id) or tp_speedj_accel_rad_s2 < 0.0:
    |         codex_autotune_wait_for_arm(campaign_epoch, trial_id, 78, candidate_token, 13, execution_profile_id, last_consumed_command_seq)
    |         campaign_epoch = read_input_integer_register(24)
    |         trial_id = read_input_integer_register(25)
    |         candidate_token = read_input_integer_register(27)
    |         execution_profile_id = read_input_integer_register(28)
    |         batch_row_index = read_input_integer_register(30)
    |         logical_batch_sequence = read_input_integer_register(31)
    |         tp_speedj_accel_rad_s2 = codex_autotune_speedj_accel(execution_profile_id)
    |         last_consumed_command_seq = read_input_integer_register(29)
    |       end
    | 
    |       codex_autotune_batch_row_echo = batch_row_index
    |       codex_autotune_logical_batch_sequence_echo = logical_batch_sequence
    |       codex_autotune_return_kind_echo = 2
    |       codex_autotune_return_guard_mask = 0
    |       codex_autotune_write_state(campaign_epoch, trial_id, 11, candidate_token, 0, execution_profile_id, last_consumed_command_seq)
    |       codex_autotune_write_state(campaign_epoch, trial_id, 20, candidate_token, 0, execution_profile_id, last_consumed_command_seq)
    |       local stop_reason = codex_step5d_autotune_trial_v1(campaign_home_pose, tp_speedj_accel_rad_s2, batch_row_index)
    |       codex_autotune_write_state(campaign_epoch, trial_id, 30, candidate_token, stop_reason, execution_profile_id, last_consumed_command_seq)
    | 
    |       if stop_reason == 2 or stop_reason == 3 or stop_reason == 17:
    |         # Transport/sensor/unsafe-entry reasons 2, 3, and 17 have no
    |         # return proof.  The no-return path never moves and never terminates
    |         # on its own.
    |         codex_autotune_wait_for_external_home(campaign_epoch, trial_id, 75, candidate_token, stop_reason, execution_profile_id, last_consumed_command_seq, campaign_home_pose, campaign_home_q)
    |         codex_autotune_write_state(campaign_epoch, trial_id, 78, candidate_token, stop_reason, execution_profile_id, last_consumed_command_seq)
    |         codex_autotune_wait_for_arm(campaign_epoch, trial_id, 78, candidate_token, stop_reason, execution_profile_id, last_consumed_command_seq)
    |       elif codex_should_auto_home(stop_reason):
    |         codex_autotune_write_state(campaign_epoch, trial_id, 40, candidate_token, stop_reason, execution_profile_id, last_consumed_command_seq)
    |         if not codex_autotune_single_owner_return(batch_row_index, campaign_home_pose, campaign_home_q):
    |           # A failed return has no Home proof.  Remain stationary and wait for
    |           # external/controller recovery before exposing READY_HOME_NEXT.
    |           codex_autotune_wait_for_external_home(campaign_epoch, trial_id, 75, candidate_token, 17, execution_profile_id, last_consumed_command_seq, campaign_home_pose, campaign_home_q)
    |         end
    |         codex_autotune_write_state(campaign_epoch, trial_id, 50, candidate_token, stop_reason, execution_profile_id, last_consumed_command_seq)
    |         codex_autotune_write_state(campaign_epoch, trial_id, 60, candidate_token, stop_reason, execution_profile_id, last_consumed_command_seq)
    | 
    |         # Every local software guard is trial-local.  The single-owner return
    |         # has already brought the robot home; publish READY_HOME_NEXT and wait
    |         # indefinitely for the next fresh ARM.  STOP/COMPLETE remain explicit
    |         # stationary shutdown commands handled by codex_autotune_wait_for_arm.
    |         codex_autotune_wait_for_arm(campaign_epoch, trial_id, 78, candidate_token, stop_reason, execution_profile_id, last_consumed_command_seq)
    |       else:
    |         # Unknown outcomes have no return proof: remain resident until an
    |         # external no-motion Home proof, then accept the next fresh ARM.
    |         codex_autotune_wait_for_external_home(campaign_epoch, trial_id, 75, candidate_token, stop_reason, execution_profile_id, last_consumed_command_seq, campaign_home_pose, campaign_home_q)
    |         codex_autotune_write_state(campaign_epoch, trial_id, 78, candidate_token, stop_reason, execution_profile_id, last_consumed_command_seq)
    |         codex_autotune_wait_for_arm(campaign_epoch, trial_id, 78, candidate_token, stop_reason, execution_profile_id, last_consumed_command_seq)
    |       end
    |     else:
    |       sync()
    |     end
    |   end
    | end
    | 
    | codex_step5d_strict_rnn_autotune_v3()
